Omron CX-Programmer project 新工程 (CX-Programmer 9.73)

# PLC 新PLC1: CP1H XA

## Global symbols (name address type ; comment)
0.00 BOOL  ; 启动
0.01 BOOL  ; 急停
100.00 BOOL  ; 欢
100.01 BOOL  ; 迎
100.02 BOOL  ; 光
100.03 BOOL  ; 临
100.04 BOOL  ; 一
100.05 BOOL  ; 汽
T0000 BOOL  ; 1步序延时
T0001 BOOL  ; 2步序延时
T0002 BOOL  ; 3步序延时
T0003 BOOL  ; 4步序延时
T0004 BOOL  ; 5步序延时
T0005 BOOL  ; 6步序延时
T0006 BOOL  ; 循环1完成延时
T0007 BOOL  ; 7步序延时
T0008 BOOL  ; 8步序延时
T0009 BOOL  ; 9步序延时
T0010 BOOL  ; 10步序延时
T0011 BOOL  ; 11步序延时
T0012 BOOL  ; 循环2完成延时
T0013 BOOL  ; 12步序延时
T0014 BOOL  ; 13步序延时
T0015 BOOL  ; 14步序延时
T0016 BOOL  ; 15步序延时
T0017 BOOL  ; 循环3完成延时
T0018 BOOL  ; 16步序延时
T0019 BOOL  ; 17步序延时
T0020 BOOL  ; 18步序延时
T0021 BOOL  ; 循环4完成延时
T0022 BOOL  ; 19步序延时
T0023 BOOL  ; 20步序延时
T0024 BOOL  ; 循环5完成延时
T0025 BOOL  ; 21步序延时
T0026 BOOL  ; 22步序结束延时
W0.00 BOOL  ; “欢”辅助输出
W0.01 BOOL  ; “欢”辅助输出
W0.02 BOOL  ; “欢”辅助输出
W0.03 BOOL  ; “欢”辅助输出
W0.04 BOOL  ; “欢”辅助输出
W0.05 BOOL  ; “欢”辅助输出
W1.00 BOOL  ; “迎”辅助输出
W1.01 BOOL  ; “迎”辅助输出
W1.02 BOOL  ; “迎”辅助输出
W1.03 BOOL  ; “迎”辅助输出
W1.04 BOOL  ; “迎”辅助输出
W1.05 BOOL  ; “迎”辅助输出
W20 CHANNEL  ; 步号
W2.00 BOOL  ; “光”辅助输出
W2.01 BOOL  ; “光”辅助输出
W2.02 BOOL  ; “光”辅助输出
W2.03 BOOL  ; “光”辅助输出
W2.04 BOOL  ; “光”辅助输出
W2.05 BOOL  ; “光”辅助输出
W3.00 BOOL  ; “临”辅助输出
W3.01 BOOL  ; “临”辅助输出
W3.02 BOOL  ; “临”辅助输出
W3.03 BOOL  ; “临”辅助输出
W3.04 BOOL  ; “临”辅助输出
W3.05 BOOL  ; “临”辅助输出
W4.00 BOOL  ; “一”辅助输出
W4.01 BOOL  ; “一”辅助输出
W4.02 BOOL  ; “一”辅助输出
W4.03 BOOL  ; “一”辅助输出
W4.04 BOOL  ; “一”辅助输出
W4.05 BOOL  ; “一”辅助输出
W5.00 BOOL  ; “汽”辅助输出
W5.01 BOOL  ; “汽”辅助输出
W5.02 BOOL  ; “汽”辅助输出
W5.03 BOOL  ; “汽”辅助输出
W5.04 BOOL  ; “汽”辅助输出
W5.05 BOOL  ; “汽”辅助输出

## Program 新程序1 (cyclic task 0)
; 这个项目包含一个广告牌灯箱控制系统，通过PLC控制器CP1H控制六个字"欢"、"迎"、"光"、"临"、"一"、"汽"的灯的亮灭，实现动态展示效果。系统使用启动按钮启动工作流程，急停按钮停止运行，使用的物理设备包括PLC控制器CP1H、广告牌灯箱、启动按钮和急停按钮。 / 按下启动按钮后，步号置为1，开始执行从1到27的步序流程。 / 步序1中，若急停按钮未按下，置位“欢”字辅助输出1。当“欢”字辅助输出置位时，点亮“欢”字灯。 / 并启动步序延时定时器1，延时10个时间单位后切换至步序2。 / 在每个步序中，仅置位相应的“欢”字辅助输出，以确保步序切换正常进行。新描述：在步序1中，置位“欢”字辅助输出1，同时其他“欢”字辅助输出2至6保持初始复位状态，以确保步序正常切换。 / 急停按钮按下时“欢”字灯立即熄灭。 / 步序2至6依次置位“迎”字辅助输出1至“汽”字辅助输出1，每次切换前等待对应步序延时定时器完成计时。当相应辅助输出置位时，点亮“迎”字灯至“汽”字灯。急停按钮按下时，所有灯光动作停止，但步号可能继续递增以维持流程记录。 / 步序7作为过渡，启动步序延时定时器7，在5个时间单位内完成计时后进入步序8，保证时序准确。 / 类似的，步序8至22通过置位和复位辅助输出实现动态灯光组合，每一步序由步序延时定时器8至22控制延时。 / 若急停按钮按下，所有灯光动作立即停止，所有灯保持熄灭状态。 / 步序23至27逐步复位所有辅助输出，确保“欢”字灯至“汽”字灯在循环结束时全部熄灭，以完成一次展示流程。

### Section 段1

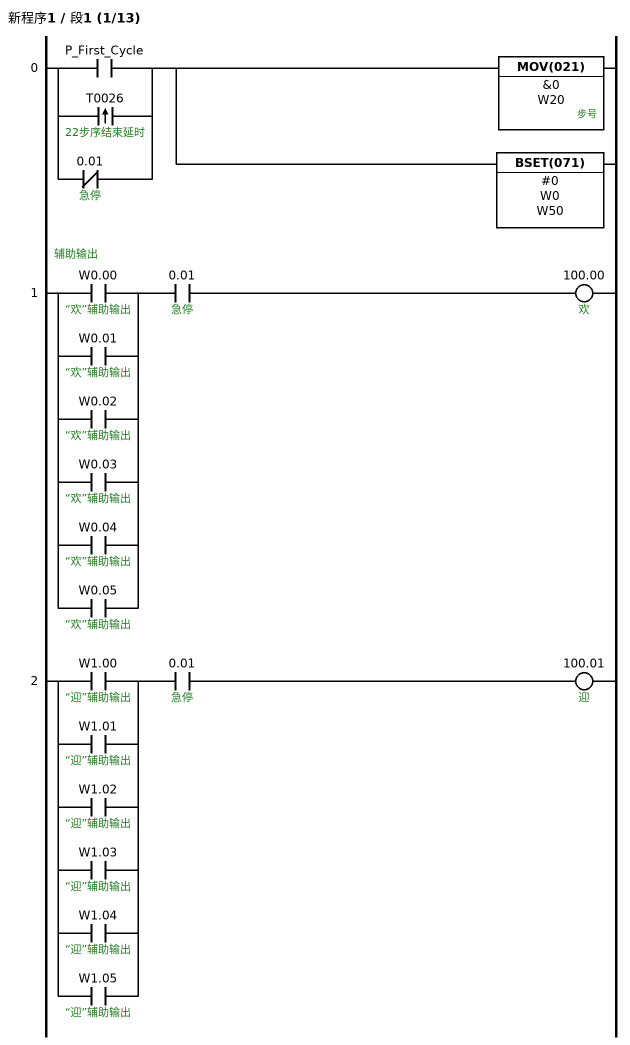
; rung 0
LD P_First_Cycle
@OR T0026  ; 22步序结束延时
ORNOT 0.01  ; 急停
MOV(021) &0 W20  ; 步号
BSET(071) #0 W0 W50
; rung 1: 辅助输出
LD W0.00  ; “欢”辅助输出
OR W0.01  ; “欢”辅助输出
OR W0.02  ; “欢”辅助输出
OR W0.03  ; “欢”辅助输出
OR W0.04  ; “欢”辅助输出
OR W0.05  ; “欢”辅助输出
AND 0.01  ; 急停
OUT 100.00  ; 欢
; rung 2
LD W1.00  ; “迎”辅助输出
OR W1.01  ; “迎”辅助输出
OR W1.02  ; “迎”辅助输出
OR W1.03  ; “迎”辅助输出
OR W1.04  ; “迎”辅助输出
OR W1.05  ; “迎”辅助输出
AND 0.01  ; 急停
OUT 100.01  ; 迎

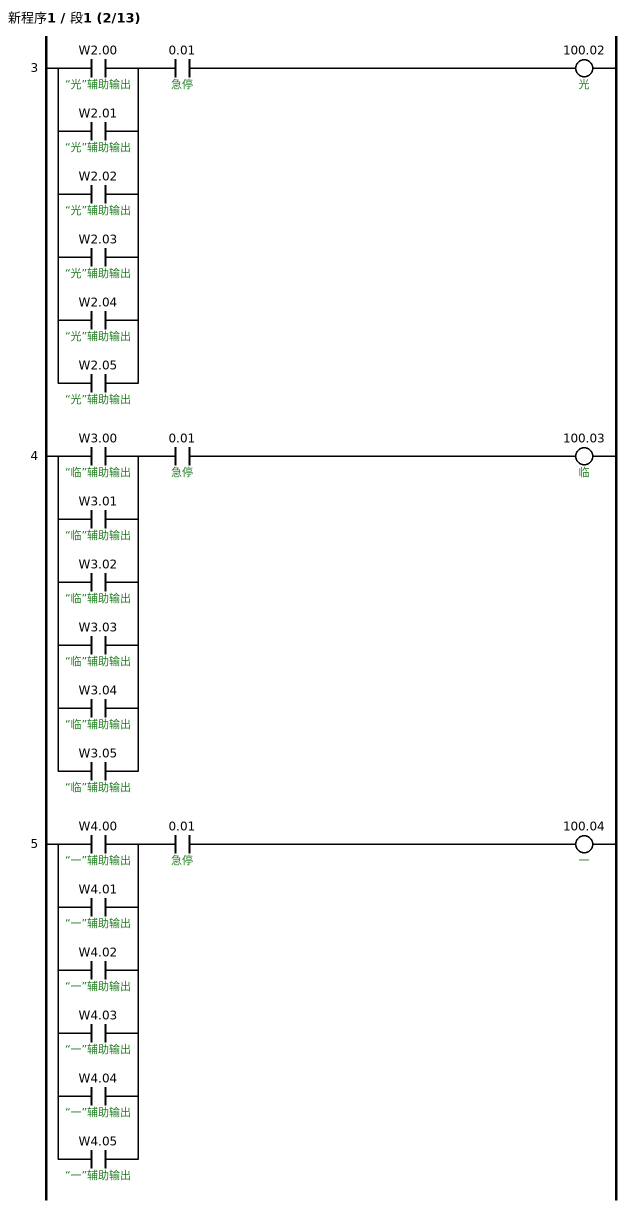
; rung 3
LD W2.00  ; “光”辅助输出
OR W2.01  ; “光”辅助输出
OR W2.02  ; “光”辅助输出
OR W2.03  ; “光”辅助输出
OR W2.04  ; “光”辅助输出
OR W2.05  ; “光”辅助输出
AND 0.01  ; 急停
OUT 100.02  ; 光
; rung 4
LD W3.00  ; “临”辅助输出
OR W3.01  ; “临”辅助输出
OR W3.02  ; “临”辅助输出
OR W3.03  ; “临”辅助输出
OR W3.04  ; “临”辅助输出
OR W3.05  ; “临”辅助输出
AND 0.01  ; 急停
OUT 100.03  ; 临
; rung 5
LD W4.00  ; “一”辅助输出
OR W4.01  ; “一”辅助输出
OR W4.02  ; “一”辅助输出
OR W4.03  ; “一”辅助输出
OR W4.04  ; “一”辅助输出
OR W4.05  ; “一”辅助输出
AND 0.01  ; 急停
OUT 100.04  ; 一

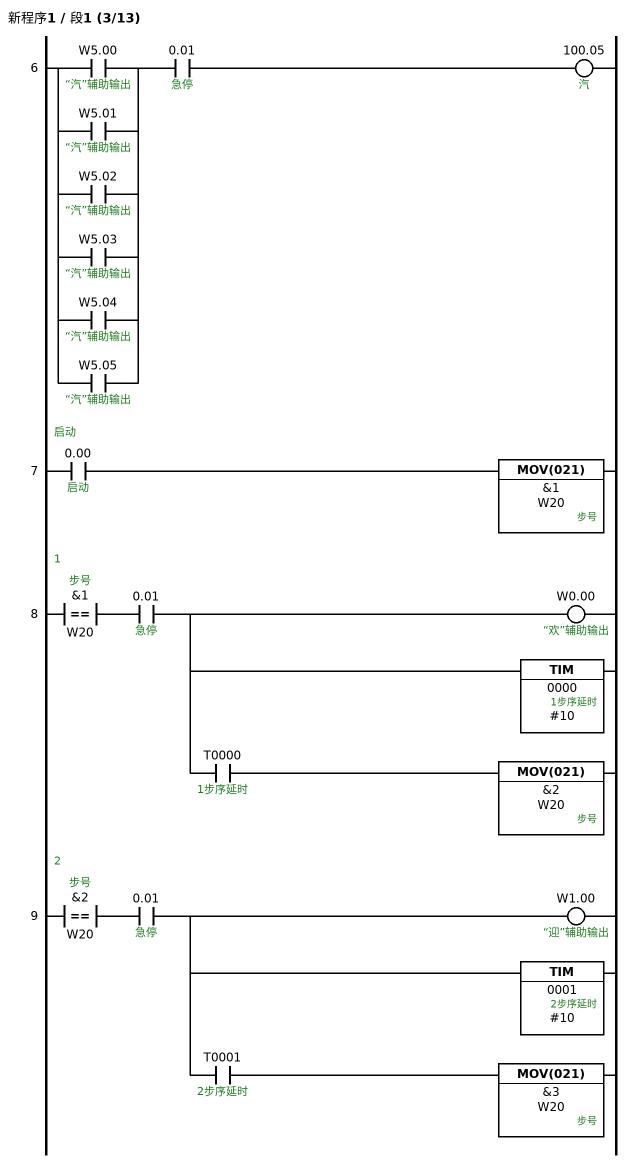
; rung 6
LD W5.00  ; “汽”辅助输出
OR W5.01  ; “汽”辅助输出
OR W5.02  ; “汽”辅助输出
OR W5.03  ; “汽”辅助输出
OR W5.04  ; “汽”辅助输出
OR W5.05  ; “汽”辅助输出
AND 0.01  ; 急停
OUT 100.05  ; 汽
; rung 7: 启动
LD 0.00  ; 启动
MOV(021) &1 W20  ; 步号
; rung 8: 1
LD=(300) &1 W20  ; 步号
AND 0.01  ; 急停
OUT W0.00  ; “欢”辅助输出
TIM 0000 #10  ; 1步序延时
AND T0000  ; 1步序延时
MOV(021) &2 W20  ; 步号
; rung 9: 2
LD=(300) &2 W20  ; 步号
AND 0.01  ; 急停
OUT W1.00  ; “迎”辅助输出
TIM 0001 #10  ; 2步序延时
AND T0001  ; 2步序延时
MOV(021) &3 W20  ; 步号

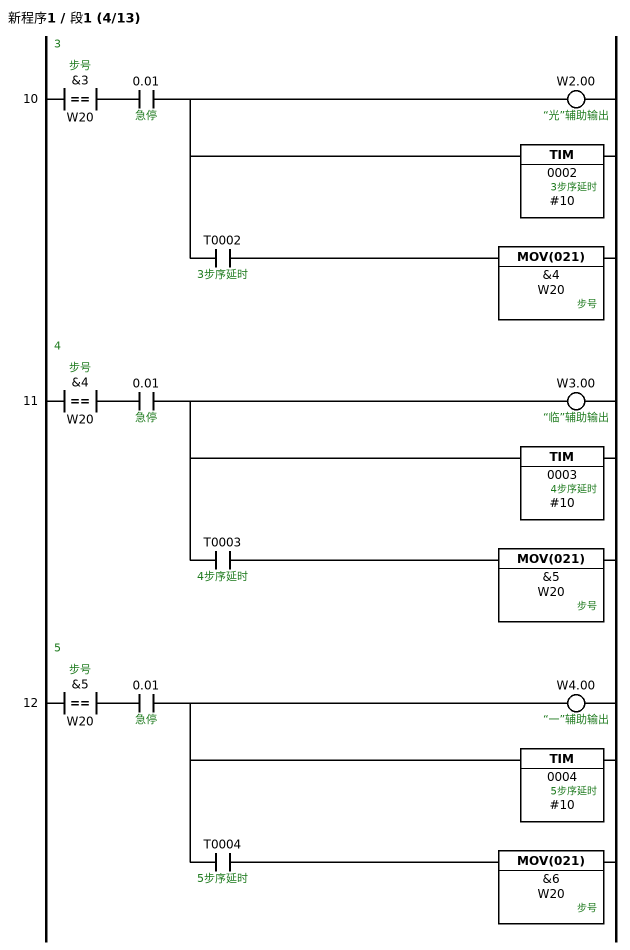
; rung 10: 3
LD=(300) &3 W20  ; 步号
AND 0.01  ; 急停
OUT W2.00  ; “光”辅助输出
TIM 0002 #10  ; 3步序延时
AND T0002  ; 3步序延时
MOV(021) &4 W20  ; 步号
; rung 11: 4
LD=(300) &4 W20  ; 步号
AND 0.01  ; 急停
OUT W3.00  ; “临”辅助输出
TIM 0003 #10  ; 4步序延时
AND T0003  ; 4步序延时
MOV(021) &5 W20  ; 步号
; rung 12: 5
LD=(300) &5 W20  ; 步号
AND 0.01  ; 急停
OUT W4.00  ; “一”辅助输出
TIM 0004 #10  ; 5步序延时
AND T0004  ; 5步序延时
MOV(021) &6 W20  ; 步号

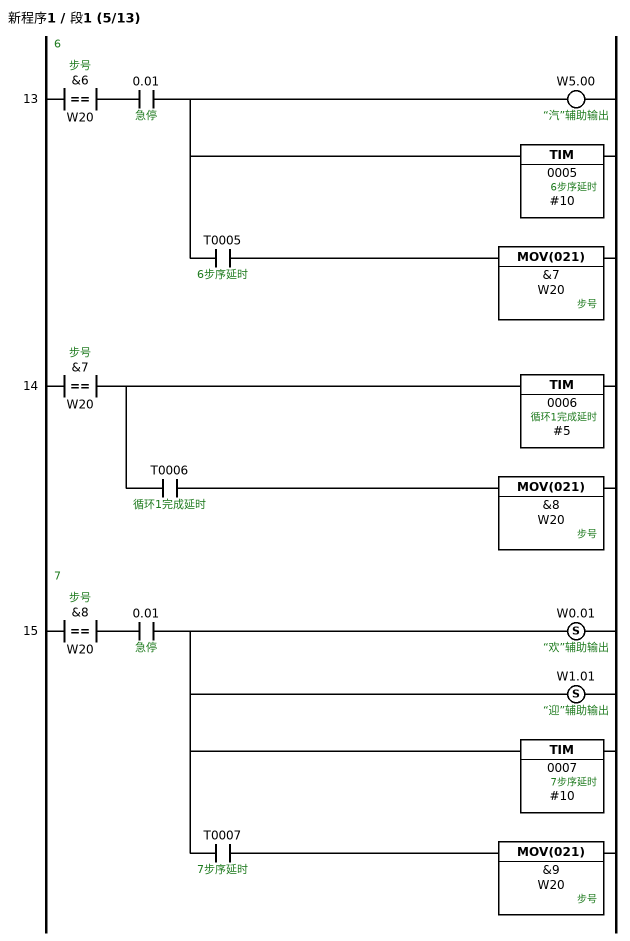
; rung 13: 6
LD=(300) &6 W20  ; 步号
AND 0.01  ; 急停
OUT W5.00  ; “汽”辅助输出
TIM 0005 #10  ; 6步序延时
AND T0005  ; 6步序延时
MOV(021) &7 W20  ; 步号
; rung 14
LD=(300) &7 W20  ; 步号
TIM 0006 #5  ; 循环1完成延时
AND T0006  ; 循环1完成延时
MOV(021) &8 W20  ; 步号
; rung 15: 7
LD=(300) &8 W20  ; 步号
AND 0.01  ; 急停
SET W0.01  ; “欢”辅助输出
SET W1.01  ; “迎”辅助输出
TIM 0007 #10  ; 7步序延时
AND T0007  ; 7步序延时
MOV(021) &9 W20  ; 步号

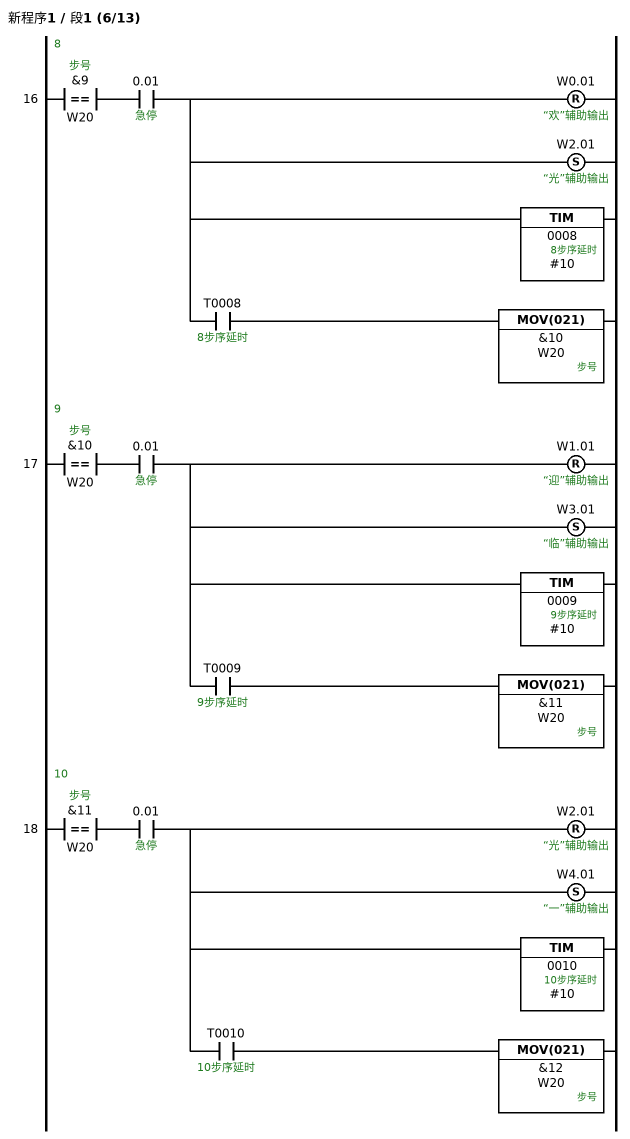
; rung 16: 8
LD=(300) &9 W20  ; 步号
AND 0.01  ; 急停
RSET W0.01  ; “欢”辅助输出
SET W2.01  ; “光”辅助输出
TIM 0008 #10  ; 8步序延时
AND T0008  ; 8步序延时
MOV(021) &10 W20  ; 步号
; rung 17: 9
LD=(300) &10 W20  ; 步号
AND 0.01  ; 急停
RSET W1.01  ; “迎”辅助输出
SET W3.01  ; “临”辅助输出
TIM 0009 #10  ; 9步序延时
AND T0009  ; 9步序延时
MOV(021) &11 W20  ; 步号
; rung 18: 10
LD=(300) &11 W20  ; 步号
AND 0.01  ; 急停
RSET W2.01  ; “光”辅助输出
SET W4.01  ; “一”辅助输出
TIM 0010 #10  ; 10步序延时
AND T0010  ; 10步序延时
MOV(021) &12 W20  ; 步号

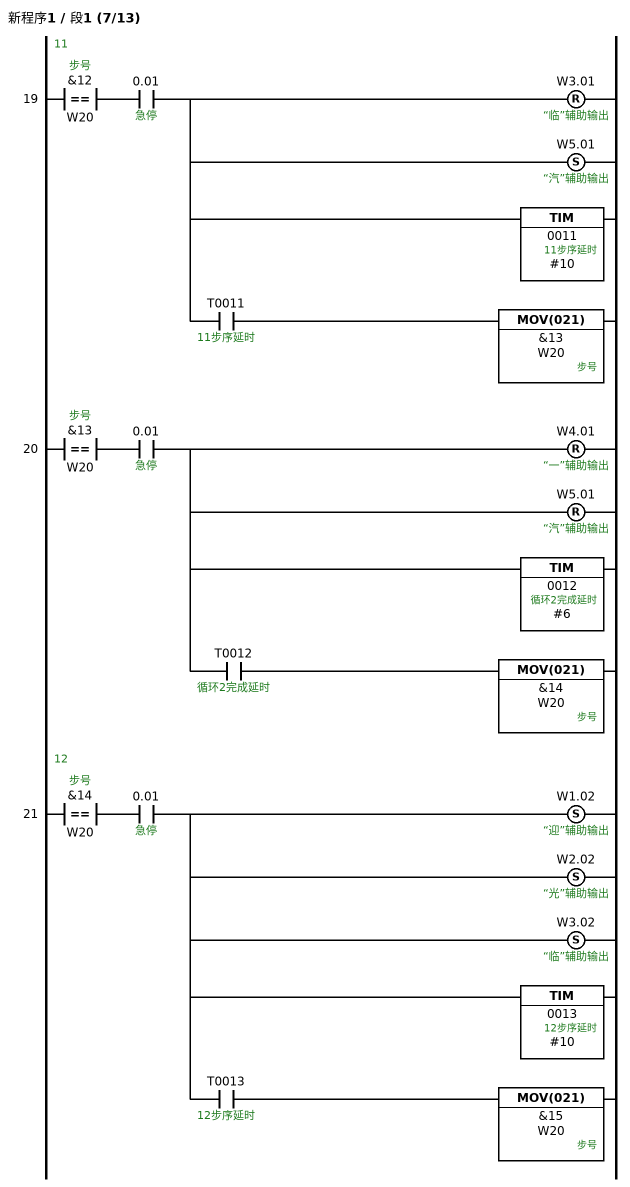
; rung 19: 11
LD=(300) &12 W20  ; 步号
AND 0.01  ; 急停
RSET W3.01  ; “临”辅助输出
SET W5.01  ; “汽”辅助输出
TIM 0011 #10  ; 11步序延时
AND T0011  ; 11步序延时
MOV(021) &13 W20  ; 步号
; rung 20
LD=(300) &13 W20  ; 步号
AND 0.01  ; 急停
RSET W4.01  ; “一”辅助输出
RSET W5.01  ; “汽”辅助输出
TIM 0012 #6  ; 循环2完成延时
AND T0012  ; 循环2完成延时
MOV(021) &14 W20  ; 步号
; rung 21: 12
LD=(300) &14 W20  ; 步号
AND 0.01  ; 急停
SET W1.02  ; “迎”辅助输出
SET W2.02  ; “光”辅助输出
SET W3.02  ; “临”辅助输出
TIM 0013 #10  ; 12步序延时
AND T0013  ; 12步序延时
MOV(021) &15 W20  ; 步号

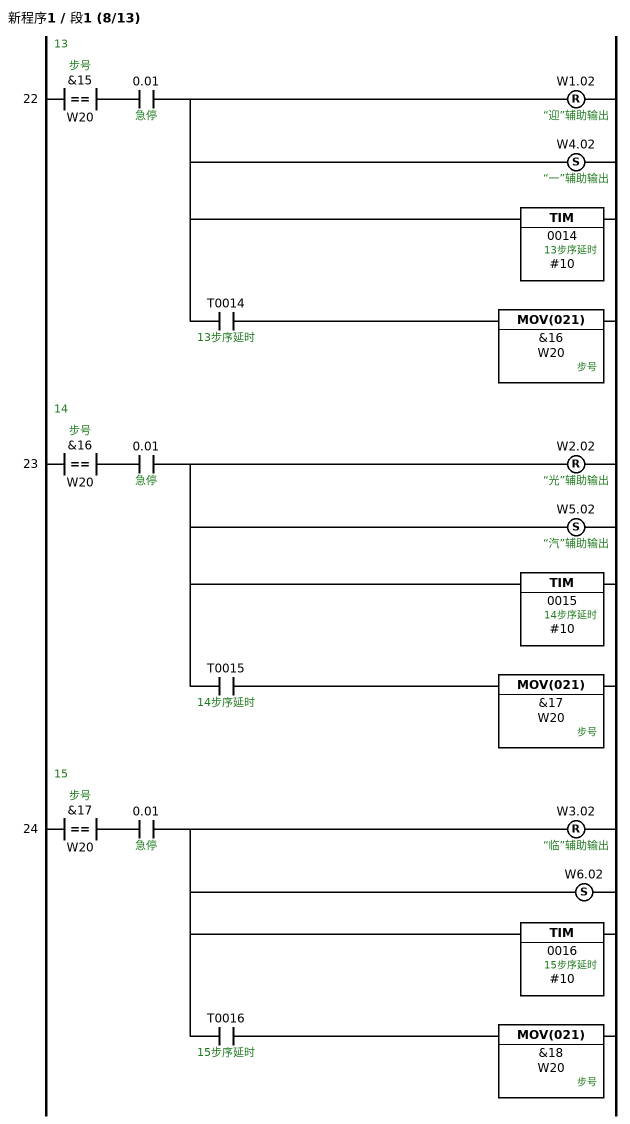
; rung 22: 13
LD=(300) &15 W20  ; 步号
AND 0.01  ; 急停
RSET W1.02  ; “迎”辅助输出
SET W4.02  ; “一”辅助输出
TIM 0014 #10  ; 13步序延时
AND T0014  ; 13步序延时
MOV(021) &16 W20  ; 步号
; rung 23: 14
LD=(300) &16 W20  ; 步号
AND 0.01  ; 急停
RSET W2.02  ; “光”辅助输出
SET W5.02  ; “汽”辅助输出
TIM 0015 #10  ; 14步序延时
AND T0015  ; 14步序延时
MOV(021) &17 W20  ; 步号
; rung 24: 15
LD=(300) &17 W20  ; 步号
AND 0.01  ; 急停
RSET W3.02  ; “临”辅助输出
SET W6.02
TIM 0016 #10  ; 15步序延时
AND T0016  ; 15步序延时
MOV(021) &18 W20  ; 步号

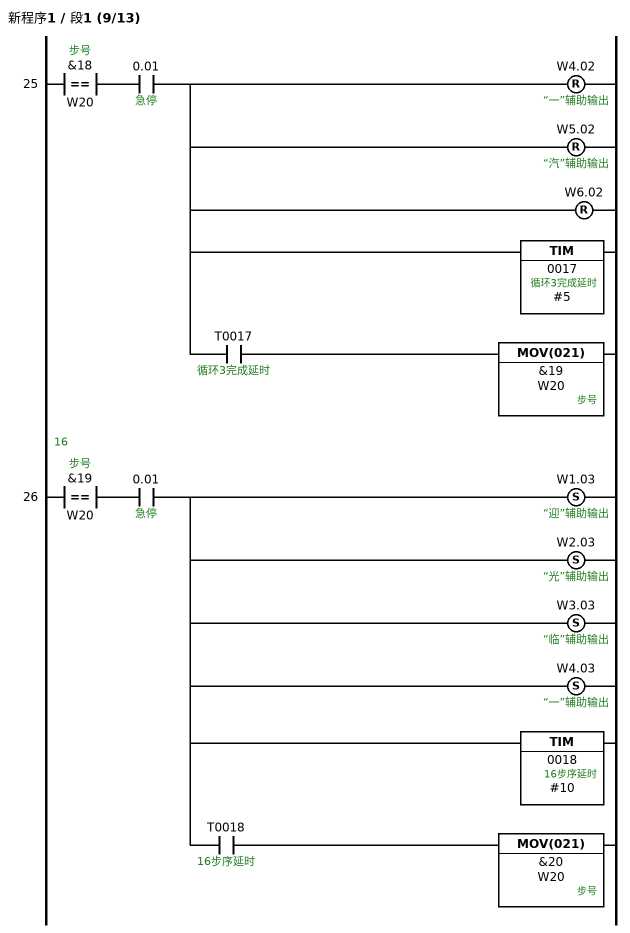
; rung 25
LD=(300) &18 W20  ; 步号
AND 0.01  ; 急停
RSET W4.02  ; “一”辅助输出
RSET W5.02  ; “汽”辅助输出
RSET W6.02
TIM 0017 #5  ; 循环3完成延时
AND T0017  ; 循环3完成延时
MOV(021) &19 W20  ; 步号
; rung 26: 16
LD=(300) &19 W20  ; 步号
AND 0.01  ; 急停
SET W1.03  ; “迎”辅助输出
SET W2.03  ; “光”辅助输出
SET W3.03  ; “临”辅助输出
SET W4.03  ; “一”辅助输出
TIM 0018 #10  ; 16步序延时
AND T0018  ; 16步序延时
MOV(021) &20 W20  ; 步号

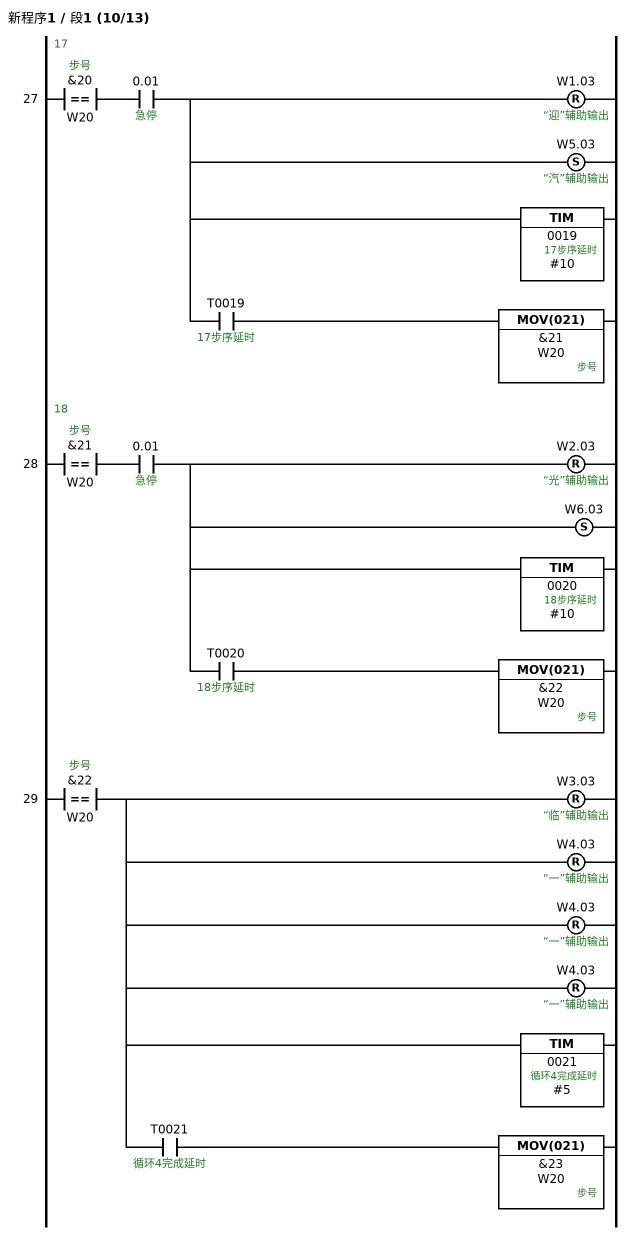
; rung 27: 17
LD=(300) &20 W20  ; 步号
AND 0.01  ; 急停
RSET W1.03  ; “迎”辅助输出
SET W5.03  ; “汽”辅助输出
TIM 0019 #10  ; 17步序延时
AND T0019  ; 17步序延时
MOV(021) &21 W20  ; 步号
; rung 28: 18
LD=(300) &21 W20  ; 步号
AND 0.01  ; 急停
RSET W2.03  ; “光”辅助输出
SET W6.03
TIM 0020 #10  ; 18步序延时
AND T0020  ; 18步序延时
MOV(021) &22 W20  ; 步号
; rung 29
LD=(300) &22 W20  ; 步号
RSET W3.03  ; “临”辅助输出
RSET W4.03  ; “一”辅助输出
RSET W4.03  ; “一”辅助输出
RSET W4.03  ; “一”辅助输出
TIM 0021 #5  ; 循环4完成延时
AND T0021  ; 循环4完成延时
MOV(021) &23 W20  ; 步号

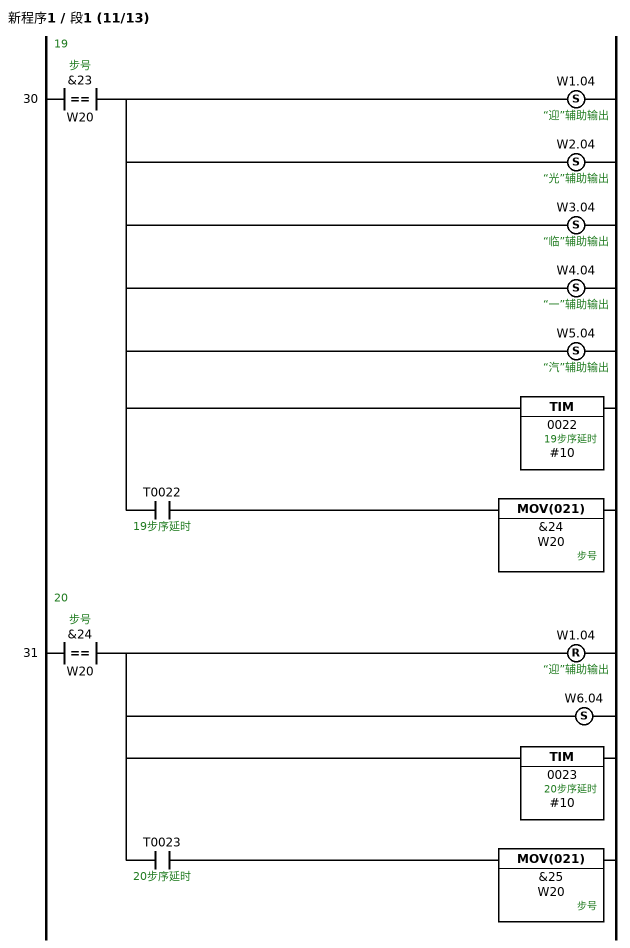
; rung 30: 19
LD=(300) &23 W20  ; 步号
SET W1.04  ; “迎”辅助输出
SET W2.04  ; “光”辅助输出
SET W3.04  ; “临”辅助输出
SET W4.04  ; “一”辅助输出
SET W5.04  ; “汽”辅助输出
TIM 0022 #10  ; 19步序延时
AND T0022  ; 19步序延时
MOV(021) &24 W20  ; 步号
; rung 31: 20
LD=(300) &24 W20  ; 步号
RSET W1.04  ; “迎”辅助输出
SET W6.04
TIM 0023 #10  ; 20步序延时
AND T0023  ; 20步序延时
MOV(021) &25 W20  ; 步号

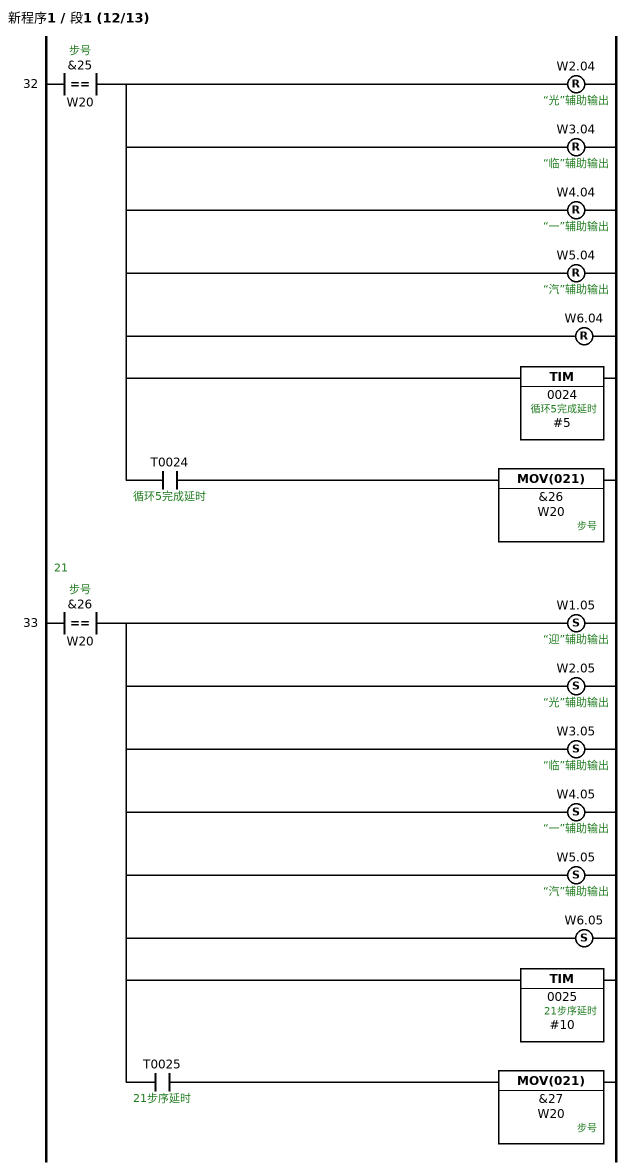
; rung 32
LD=(300) &25 W20  ; 步号
RSET W2.04  ; “光”辅助输出
RSET W3.04  ; “临”辅助输出
RSET W4.04  ; “一”辅助输出
RSET W5.04  ; “汽”辅助输出
RSET W6.04
TIM 0024 #5  ; 循环5完成延时
AND T0024  ; 循环5完成延时
MOV(021) &26 W20  ; 步号
; rung 33: 21
LD=(300) &26 W20  ; 步号
SET W1.05  ; “迎”辅助输出
SET W2.05  ; “光”辅助输出
SET W3.05  ; “临”辅助输出
SET W4.05  ; “一”辅助输出
SET W5.05  ; “汽”辅助输出
SET W6.05
TIM 0025 #10  ; 21步序延时
AND T0025  ; 21步序延时
MOV(021) &27 W20  ; 步号

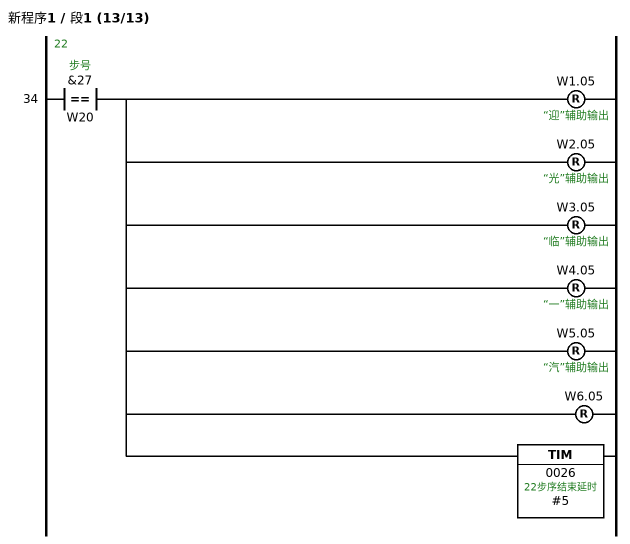
; rung 34: 22
LD=(300) &27 W20  ; 步号
RSET W1.05  ; “迎”辅助输出
RSET W2.05  ; “光”辅助输出
RSET W3.05  ; “临”辅助输出
RSET W4.05  ; “一”辅助输出
RSET W5.05  ; “汽”辅助输出
RSET W6.05
TIM 0026 #5  ; 22步序结束延时

### Section END
; rung 0
END(001)